FUNCTION_BLOCK FB_CylinderCutX EXTENDS FB_ComponentBase IMPLEMENTS I_Cylinder
VAR
    
    _ExtendRequestX  : BOOL;
    _RetractRequestX : BOOL;
    _ExtendedX       : BOOL;
    _RetractedX      : BOOL;
    _ExtendingX      : BOOL;
    _RetractingX     : BOOL;
	




    Extend_RTRIG  : R_TRIG;
    Retract_RTRIG : R_TRIG;

    //HMI 
    Cylinder_HMI : ST_Cylinder_HMI;
	

    MovementTimer : TON;
    

    CylinderAlarms : ARRAY[1..3] OF FB_TcAlarm;
END_VAR

VAR_INPUT
   	CylinderSensorCutX 			AT%I*		:	BOOL;
END_VAR

VAR_OUTPUT
	CylinderValveCutX			AT%Q*		:	BOOL;
END_VAR

PROPERTY Config : ST_Cylinder_Config
GET
Config := Cylinder_HMI.Config;
END_GET
SET
Cylinder_HMI.Config := Config;
END_SET
END_PROPERTY

METHOD PROTECTED CreateEvents
VAR_INPUT
END_VAR
SUPER^.CreateEvents();

// Powiązanie tablicy alarmów z klasą CylinderAlarms z TMC
F_CreateAllEventsInClass(
    Alarms     := CylinderAlarms,
    ClassSize  := SIZEOF(TC_EVENTS.CylinderAlarms),
    pInitEvent := ADR(TC_EVENTS.CylinderAlarms.InitReferenceEvent),
    Prefix     := _Name
);


SUPER^.CreateEvents();
END_METHOD

METHOD CyclicLogic
// One shot the requests
Extend_RTRIG(CLK := _ExtendRequestX);
Retract_RTRIG(CLK := _RetractRequestX);

// Handle Extend
IF Extend_RTRIG.Q THEN
    CylinderValveCutX := TRUE;
    _ExtendingX       := TRUE;
    _RetractingX      := FALSE;
    _RetractedX       := FALSE;
    _RetractRequestX  := FALSE;
END_IF

// Handle Retract
IF Retract_RTRIG.Q THEN
    CylinderValveCutX := FALSE;
    _ExtendingX       := FALSE;
    _RetractingX      := TRUE;
    _ExtendedX        := FALSE;
    _ExtendRequestX   := FALSE;
END_IF

// Aktualizacja stanu wyłącznie z czujnika
_ExtendedX  := CylinderSensorCutX;
_RetractedX := NOT CylinderSensorCutX;

// Status ruchu – tylko gdy trwa przejście
_ExtendingX  := _ExtendingX  AND NOT _ExtendedX;
_RetractingX := _RetractingX AND NOT _RetractedX;

// Odmierzanie czasu ruchu (używamy SEL żeby brać czas wysuwu lub chowania)
MovementTimer(
    IN := _ExtendingX OR _RetractingX,
    PT := LREAL_TO_TIME(SEL(_ExtendingX, Cylinder_HMI.Config.RetractTimeX, Cylinder_HMI.Config.ExtendTimeX) * 1000.0) 
);

// Wywołanie logiki bazowej komponentu (Tylko raz!)
SUPER^.CyclicLogic();

// Aktualizacja najwyższego priorytetu błędu dla komponentu
_CurrentAlarmSeverity := F_GetMaxSeverityRaised(Alarms := CylinderAlarms, CurrentSeverity := _CurrentAlarmSeverity);
END_METHOD

PROPERTY Error : BOOL
GET
Error := _Error;
END_GET
SET
_Error := Error;
END_SET
END_PROPERTY

METHOD Extend
_ExtendRequestX  := TRUE;
_RetractRequestX := FALSE;
END_METHOD

PROPERTY Extended : BOOL
GET
Extended := _ExtendedX;
END_GET
END_PROPERTY

METHOD PROTECTED HMICommunication
VAR_INPUT
END_VAR
SUPER^.HMICommunication();

//Handle the requests to extend and retract
IF ComponentBase_HMI.Status.HMIControlAvailable THEN
    IF Cylinder_HMI.Command.RetractExtendX THEN
        Extend();
    ELSIF Cylinder_HMI.Command.RetractCylinderX THEN
        Retract();
    END_IF
END_IF

//Update HMI status info
Cylinder_HMI.Status.ExtendedX    := _ExtendedX;
Cylinder_HMI.Status.ExtendingX   := _ExtendingX;
Cylinder_HMI.Status.RetractedX   := _RetractedX;
Cylinder_HMI.Status.RetractingX  := _RetractingX;
END_METHOD

//! @summary Basic component initialization logic
METHOD PROTECTED Initialize : BOOL;

//! @description This method is called by <c>CyclicLogic()</c> as required

IF CylinderSensorCutX THEN
    _ExtendedX  := TRUE;
    _RetractedX := FALSE;
ELSE
    _ExtendedX  := FALSE;
    _RetractedX := TRUE;
END_IF

_ExtendingX      := FALSE;
_ExtendRequestX  := FALSE;
_RetractingX     := FALSE;
_RetractRequestX := FALSE;

Initialize := SUPER^.Initialize();
END_METHOD

METHOD PROTECTED Monitoring
VAR_INPUT
END_VAR
_Busy := _ExtendingX OR _RetractingX;

// Jeśli czas minął, zgłoś odpowiedni błąd
IF MovementTimer.Q THEN
    _Error   := TRUE;
    _ErrorID := 1; 


    IF _ExtendingX AND NOT CylinderAlarms[E_CylinderAlarms.ExtendTimeout].bRaised THEN
        RaiseAlarmWithStrings(CylinderAlarms[E_CylinderAlarms.ExtendTimeout], '', '');
    
    ELSIF _RetractingX AND NOT CylinderAlarms[E_CylinderAlarms.RetractTimeout].bRaised THEN
        RaiseAlarmWithStrings(CylinderAlarms[E_CylinderAlarms.RetractTimeout], '', '');
    END_IF
END_IF

SUPER^.Monitoring();
END_METHOD

METHOD Retract
_ExtendRequestX  := FALSE;
_RetractRequestX := TRUE;
END_METHOD

PROPERTY Retracted : BOOL
GET
Retracted := _RetractedX;
END_GET
END_PROPERTY

END_FUNCTION_BLOCK

(* stored: Version 1.1.0.1, ProductVersion 3.1.4024.15
   POU FB_CylinderCutX: Id {264d7628-92d6-4793-ab2e-0fdd41979bbf}, SpecialFunc None
   Folder I_ComponentBase: Id {f559450c-ac92-42b8-948d-4319dcd66586}
   Folder I_CyclicFB: Id {06d0f814-9e61-4022-8b49-954679eac850}
   Folder I_Cylinder: Id {23231c33-e76f-4db7-9535-6a6ba8d8bb21}
   Property Config: Id {8e55ac5e-2dfd-4a5e-9f25-bccf0149b5ca}
   Get Get: Id {05aef8fe-7f7f-4070-82a6-dec38d6a2d49}
   Set Set: Id {967226d9-3fe4-4d93-9507-0c4574cc811f}
   Method CreateEvents: Id {b37c1c7a-2ee5-4bc0-bd63-7a1bd375f4f8}
   Method CyclicLogic: Id {9cd1ea00-8a5e-4fbd-a921-2bb3db34198f}
   Property Error: Id {4b52a11a-b99a-4897-8ac1-f2337615a2fb}
   Get Get: Id {398673bb-dff0-47bd-ab7b-b29e5718d541}
   Set Set: Id {1d245d19-063a-4b5f-823e-b0c571aa60c0}
   Method Extend: Id {ddb1a4c0-2458-4226-b284-f5ac382d347c}
   Property Extended: Id {1eb0eef5-7872-4e02-b38c-f05cddbbc353}
   Get Get: Id {88ee6066-a111-4e25-836f-5aab3305bf2e}
   Method HMICommunication: Id {b22c0ddf-b951-40f3-9594-3d06c6305168}
   Method Initialize: Id {ba8ff5ec-04c4-4da9-9ad0-5df11ced28f9}
   Method Monitoring: Id {8ba17133-ef6f-49ff-9719-2b67cb73a455}
   Method Retract: Id {9cc3c678-2df3-46c2-9291-f83f618c1985}
   Property Retracted: Id {c9e67c1e-2567-4eaa-a173-7c4db4a9f724}
   Get Get: Id {9d70c136-c25b-4efd-b8d4-0f770186e108} *)
